Fanuc KAREL source: kt00635.KL

-- PROVISIONAL review KL for V1013-1; original PC SHA256 590b6e08ab99e074bea3a42fe811f6097b95a0d753920469a6f2e71407834992
-- Incomplete behavior may be omitted. Consult companion uncertainty JSON. Do not deploy.
PROGRAM KT00635
%NOLOCKGROUP
VAR
  OUT : REAL
-- UNRESOLVED_DECL Y1 type=002018
-- UNRESOLVED_DECL Y2 type=002018
BEGIN
  -- UNRESOLVED_PC offsets 5-19; opcodes 2E,22,9D,33,B2
  -- UNRESOLVED_PC offsets 24-38; opcodes 2E,22,9D,33,B2
  -- UNRESOLVED_PC offsets 43-57; opcodes 2E,22,9D,33,B2
  -- UNRESOLVED_PC offsets 62-76; opcodes 2E,22,9D,33,B2
  -- UNRESOLVED_PC offsets 81-98; opcodes 22,9D,33,B1,48,64,23
  -- UNRESOLVED_PC offsets 103-107; opcodes 7F
END KT00635
